TYPE T_Ctrl_SIf_MOD_Out :
STRUCT
	/// Ready Signal
	bolReady: BASE_PLC.T_Ctrl_IoBool;
END_STRUCT
END_TYPE

(* stored: Version 1.1.0.1, ProductVersion 3.1.0.25
   DUT T_Ctrl_SIf_MOD_Out: Id {08e402dd-7973-47f5-b63b-307e53430d30} *)
